Yaskawa INFORM job: ramp_planes_program.JBI

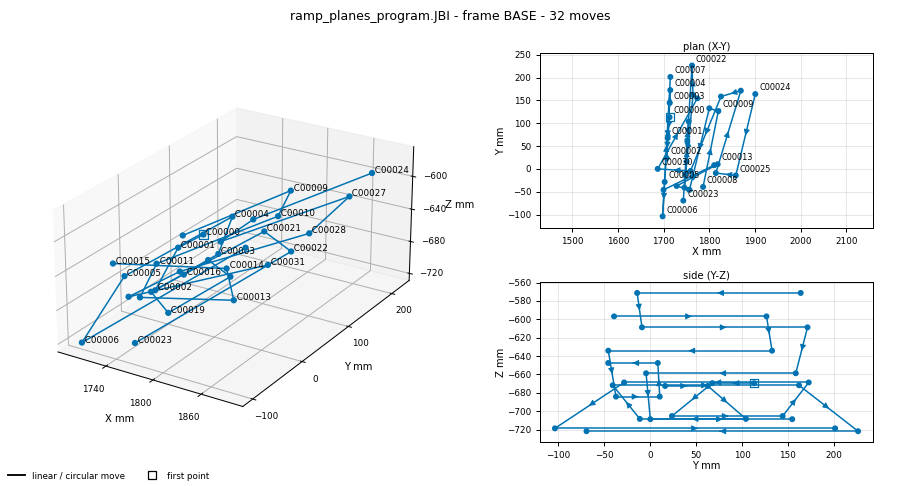
[picture p0: tool path of ramp_planes_program.JBI in frame BASE, 32 of 38 moves have a stored position in this frame; points joined in program order, loops and branches not executed]
/JOB
//NAME ramp_planes_program
//POS
///NPOS 32,0,32,0,0,0
///TOOL 0
///POSTYPE BASE
///RECTAN
///RCONF 0,0,0,0,0,0,0,0,0,0,0,0,0,0,0,0,0,0,0,0,0,0,0,0
C00000=1713.152300,113.303630,-669.533780,-175.000000,-88.858308,-5.000000
C00001=1708.992300,67.671990,-669.533780,-175.000000,-88.858308,-5.000000
C00002=1706.932300,23.758690,-705.329280,-175.000000,-88.858308,-5.000000
C00003=1713.382300,144.285490,-705.329280,-175.000000,-88.858308,-5.000000
C00004=1714.672300,172.690790,-668.726740,180.000000,-60.000000,0.000000
C00005=1702.472300,-28.301110,-668.726740,180.000000,-60.000000,0.000000
C00006=1697.962300,-103.631110,-718.726740,180.000000,-60.000000,0.000000
C00007=1714.892300,201.358290,-718.726740,180.000000,-60.000000,0.000000
C00008=1786.423630,-39.257900,-596.809650,175.000000,-59.685961,-5.000000
C00009=1819.862000,126.692100,-596.809650,175.000000,-59.685961,-5.000000
C00010=1800.088650,132.752100,-634.189150,175.000000,-59.685961,-5.000000
C00011=1756.740900,-45.537900,-634.189150,175.000000,-59.685961,-5.000000
C00012=1728.599600,-37.167900,-684.189150,175.000000,-59.685961,-5.000000
C00013=1818.454800,10.462100,-684.189150,175.000000,-59.685961,-5.000000
C00014=1810.719600,8.372100,-647.586610,180.000000,-60.000000,0.000000
C00015=1699.957400,-45.627900,-647.586610,180.000000,-60.000000,0.000000
C00016=1750.330600,16.295845,-672.576910,175.000000,-89.584182,-5.000000
C00017=1752.050600,62.820895,-672.576910,175.000000,-89.584182,-5.000000
C00018=1754.990600,104.302695,-708.425410,175.000000,-89.584182,-5.000000
C00019=1747.680600,-11.225505,-708.425410,175.000000,-89.584182,-5.000000
C00020=1745.640600,-40.718005,-671.822869,180.000000,-60.000000,0.000000
C00021=1764.350600,162.062595,-671.822869,180.000000,-60.000000,0.000000
C00022=1762.320600,226.373595,-721.822869,180.000000,-60.000000,0.000000
C00023=1743.200600,-69.282205,-721.822869,180.000000,-60.000000,0.000000
C00024=1900.692050,163.927855,-571.298800,175.000000,-47.732091,-5.000000
C00025=1858.051850,-14.152145,-571.298800,175.000000,-47.732091,-5.000000
C00026=1814.339550,-8.872145,-608.742300,175.000000,-47.732091,-5.000000
C00027=1869.022850,171.347855,-608.742300,175.000000,-47.732091,-5.000000
C00028=1825.658550,158.567855,-658.742300,175.000000,-47.732091,-5.000000
C00029=1758.915150,-4.422145,-658.742300,175.000000,-47.732091,-5.000000
C00030=1687.196150,0.227855,-708.742300,175.000000,-47.732091,-5.000000
C00031=1773.888150,154.687855,-708.742300,175.000000,-47.732091,-5.000000
///POSTYPE PULSE
///PULSE
EC00000=0
EC00001=0
EC00002=0
EC00003=0
EC00004=0
EC00005=0
EC00006=0
EC00007=0
EC00008=92160
EC00009=92160
EC00010=92160
EC00011=92160
EC00012=92160
EC00013=92160
EC00014=92160
EC00015=92160
EC00016=184320
EC00017=184320
EC00018=184320
EC00019=184320
EC00020=184320
EC00021=184320
EC00022=184320
EC00023=184320
EC00024=276480
EC00025=276480
EC00026=276480
EC00027=276480
EC00028=276480
EC00029=276480
EC00030=276480
EC00031=276480
//INST
///DATE 2023/08/07 12:52
///ATTR SC,RW,RJ
////FRAME BASE
///GROUP1 RB1,ST1
NOP
MOVJ P009 EX000 VJ=15.00
MOVJ P009 VJ=15.00
MOVJ C00000 EC00000 VJ=15.0
CALL JOB:SPYON
MOVL C00001 EC00001 V=150.0
MOVL C00002 EC00002 V=150.0
MOVL C00003 EC00003 V=150.0
MOVL C00004 EC00004 V=150.0
MOVL C00005 EC00005 V=150.0
MOVL C00006 EC00006 V=150.0
MOVL C00007 EC00007 V=150.0
CALL JOB:SPYOF
MOVJ P009 VJ=15.00
MOVJ C00008 EC00008 VJ=15.0
CALL JOB:SPYON
MOVL C00009 EC00009 V=150.0
MOVL C00010 EC00010 V=150.0
MOVL C00011 EC00011 V=150.0
MOVL C00012 EC00012 V=150.0
MOVL C00013 EC00013 V=150.0
MOVL C00014 EC00014 V=150.0
MOVL C00015 EC00015 V=150.0
CALL JOB:SPYOF
MOVJ P009 VJ=15.00
MOVJ C00016 EC00016 VJ=15.0
CALL JOB:SPYON
MOVL C00017 EC00017 V=150.0
MOVL C00018 EC00018 V=150.0
MOVL C00019 EC00019 V=150.0
MOVL C00020 EC00020 V=150.0
MOVL C00021 EC00021 V=150.0
MOVL C00022 EC00022 V=150.0
MOVL C00023 EC00023 V=150.0
CALL JOB:SPYOF
MOVJ P009 VJ=15.00
MOVJ C00024 EC00024 VJ=15.0
CALL JOB:SPYON
MOVL C00025 EC00025 V=150.0
MOVL C00026 EC00026 V=150.0
MOVL C00027 EC00027 V=150.0
MOVL C00028 EC00028 V=150.0
MOVL C00029 EC00029 V=150.0
MOVL C00030 EC00030 V=150.0
MOVL C00031 EC00031 V=150.0
CALL JOB:SPYOF
MOVJ P009 VJ=15.00
END
